(* PLC project Untitled1, Beckhoff Automation GmbH TwinCAT PLC Control 3.5.13.20 *)
(* stored: creationDateTime 2022-07-20T15:22:57.6890224, modificationDateTime 2022-07-20T15:22:57.6890224 *)

{attribute 'qualified_only'}
{attribute 'strict'}
TYPE eFirmerVendorEvent2 : (eNoInfo := 0, ePowerLimitationForHighTemperature := 1, ePowerLimitationForHighDCVoltage := 2, ePowerLimitationFromCapabilityRating := 3);
END_TYPE
